PROGRAM MAIN
VAR
END_VAR

END_PROGRAM

(* stored: Version 1.1.0.1
   POU MAIN: Id {9ec2eaa1-3caf-449d-ba9b-1ecd3852b5f2}, SpecialFunc None *)
